FUNCTION_BLOCK E_TP (* standard timer function block (pulse) *)
  (* Standard: 61499-2; Classification: standard timer function block; Description: Copyright (c) 2024 HR Agrartechnik GmbH This program and the accompanying materials are made available under the terms of the Eclipse Public License 2.0 which is available at https://www.eclipse.org/legal/epl-2.0/ SPDX-License-Identifier: EPL-2.0 *)
  (* Version 1.0, 2024-03-04, Franz Hoepfinger, HR Agrartechnik GmbH *)
  (* Version 1.1, 2024-04-23, Franz Hoepfinger, HR Agrartechnik GmbH, Add a Reset to Timer FBs *)
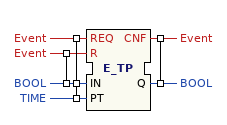
  EVENT_INPUT
    REQ WITH IN, PT; (* Service Request *)
    R WITH IN; (* Reset *)
  END_EVENT
  EVENT_OUTPUT
    CNF WITH Q; (* Confirmation of Requested Service *)
  END_EVENT
  VAR_INPUT
    IN : BOOL; (* Input *)
    PT : TIME; (* Pulse time *)
  END_VAR
  VAR_OUTPUT
    Q : BOOL; (* Output *)
  END_VAR
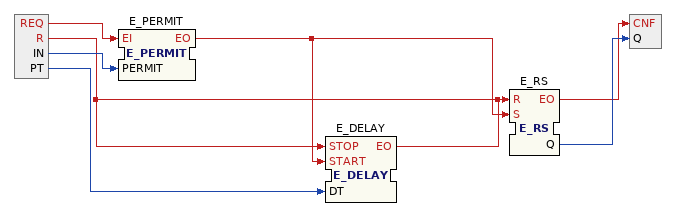
  FBS
    E_DELAY : E_DELAY;
    E_RS : E_RS;
    E_PERMIT : E_PERMIT;
  END_FBS
  EVENT_CONNECTIONS
    E_RS.EO TO CNF;
    R TO E_DELAY.STOP;
    R TO E_RS.R;
    E_DELAY.EO TO E_RS.R;
    REQ TO E_PERMIT.EI;
    E_PERMIT.EO TO E_RS.S;
    E_PERMIT.EO TO E_DELAY.START;
  END_CONNECTIONS
  DATA_CONNECTIONS
    PT TO E_DELAY.DT;
    E_RS.Q TO Q;
    IN TO E_PERMIT.PERMIT;
  END_CONNECTIONS
END_FUNCTION_BLOCK
